// TIA Portal V20 export
FUNCTION "CallCycleTimerMapping" : Void   // FC32781, LAD
// stored: SetENOAutomatically false
   VAR CONSTANT
      TRUE : Bool := TRUE;
   END_VAR
BEGIN

REGION Network 1: cycleTimerDataSet[1]
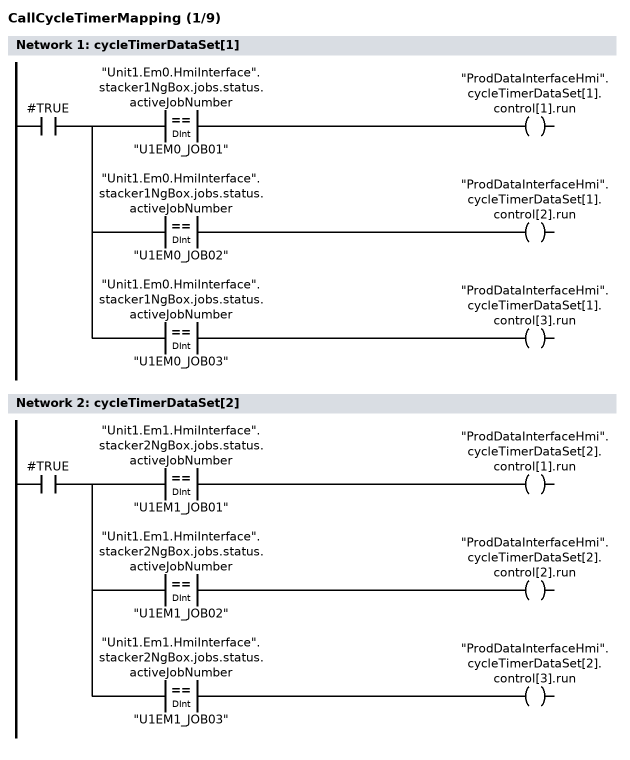
   RUNG wire#powerrail
      Contact( #TRUE )
      wire#w1
      { S7_Templates := "SrcType := DInt" } EQ_Contact(in1 := "Unit1.Em0.HmiInterface".stacker1NgBox.jobs.status.activeJobNumber, in2 := "U1EM0_JOB01")
      Coil( "ProdDataInterfaceHmi".cycleTimerDataSet[1].control[1].run )
   END_RUNG
   RUNG wire#w1
      { S7_Templates := "SrcType := DInt" } EQ_Contact(in1 := "Unit1.Em0.HmiInterface".stacker1NgBox.jobs.status.activeJobNumber, in2 := "U1EM0_JOB02")
      Coil( "ProdDataInterfaceHmi".cycleTimerDataSet[1].control[2].run )
   END_RUNG
   RUNG wire#w1
      { S7_Templates := "SrcType := DInt" } EQ_Contact(in1 := "Unit1.Em0.HmiInterface".stacker1NgBox.jobs.status.activeJobNumber, in2 := "U1EM0_JOB03")
      Coil( "ProdDataInterfaceHmi".cycleTimerDataSet[1].control[3].run )
   END_RUNG
   // the same network as SCL:
   "ProdDataInterfaceHmi".cycleTimerDataSet[1].control[1].run := #TRUE AND ("Unit1.Em0.HmiInterface".stacker1NgBox.jobs.status.activeJobNumber = "U1EM0_JOB01");
   "ProdDataInterfaceHmi".cycleTimerDataSet[1].control[2].run := #TRUE AND ("Unit1.Em0.HmiInterface".stacker1NgBox.jobs.status.activeJobNumber = "U1EM0_JOB02");
   "ProdDataInterfaceHmi".cycleTimerDataSet[1].control[3].run := #TRUE AND ("Unit1.Em0.HmiInterface".stacker1NgBox.jobs.status.activeJobNumber = "U1EM0_JOB03");
END_REGION

REGION Network 2: cycleTimerDataSet[2]
   RUNG wire#powerrail
      Contact( #TRUE )
      wire#w1
      { S7_Templates := "SrcType := DInt" } EQ_Contact(in1 := "Unit1.Em1.HmiInterface".stacker2NgBox.jobs.status.activeJobNumber, in2 := "U1EM1_JOB01")
      Coil( "ProdDataInterfaceHmi".cycleTimerDataSet[2].control[1].run )
   END_RUNG
   RUNG wire#w1
      { S7_Templates := "SrcType := DInt" } EQ_Contact(in1 := "Unit1.Em1.HmiInterface".stacker2NgBox.jobs.status.activeJobNumber, in2 := "U1EM1_JOB02")
      Coil( "ProdDataInterfaceHmi".cycleTimerDataSet[2].control[2].run )
   END_RUNG
   RUNG wire#w1
      { S7_Templates := "SrcType := DInt" } EQ_Contact(in1 := "Unit1.Em1.HmiInterface".stacker2NgBox.jobs.status.activeJobNumber, in2 := "U1EM1_JOB03")
      Coil( "ProdDataInterfaceHmi".cycleTimerDataSet[2].control[3].run )
   END_RUNG
   // the same network as SCL:
   "ProdDataInterfaceHmi".cycleTimerDataSet[2].control[1].run := #TRUE AND ("Unit1.Em1.HmiInterface".stacker2NgBox.jobs.status.activeJobNumber = "U1EM1_JOB01");
   "ProdDataInterfaceHmi".cycleTimerDataSet[2].control[2].run := #TRUE AND ("Unit1.Em1.HmiInterface".stacker2NgBox.jobs.status.activeJobNumber = "U1EM1_JOB02");
   "ProdDataInterfaceHmi".cycleTimerDataSet[2].control[3].run := #TRUE AND ("Unit1.Em1.HmiInterface".stacker2NgBox.jobs.status.activeJobNumber = "U1EM1_JOB03");
END_REGION

REGION Network 3: cycleTimerDataSet[3]
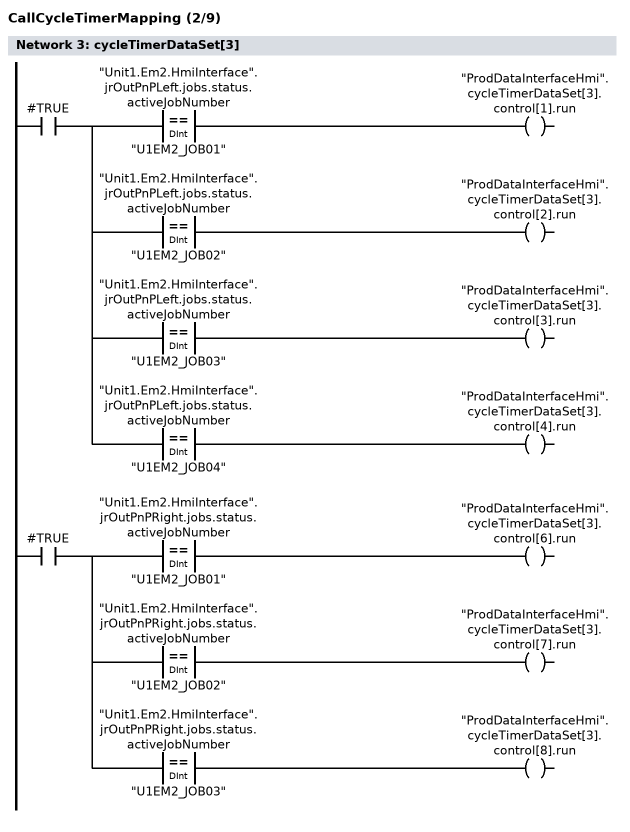
   RUNG wire#powerrail
      Contact( #TRUE )
      wire#w1
      { S7_Templates := "SrcType := DInt" } EQ_Contact(in1 := "Unit1.Em2.HmiInterface".jrOutPnPLeft.jobs.status.activeJobNumber, in2 := "U1EM2_JOB01")
      Coil( "ProdDataInterfaceHmi".cycleTimerDataSet[3].control[1].run )
   END_RUNG
   RUNG wire#w1
      { S7_Templates := "SrcType := DInt" } EQ_Contact(in1 := "Unit1.Em2.HmiInterface".jrOutPnPLeft.jobs.status.activeJobNumber, in2 := "U1EM2_JOB02")
      Coil( "ProdDataInterfaceHmi".cycleTimerDataSet[3].control[2].run )
   END_RUNG
   RUNG wire#w1
      { S7_Templates := "SrcType := DInt" } EQ_Contact(in1 := "Unit1.Em2.HmiInterface".jrOutPnPLeft.jobs.status.activeJobNumber, in2 := "U1EM2_JOB03")
      Coil( "ProdDataInterfaceHmi".cycleTimerDataSet[3].control[3].run )
   END_RUNG
   RUNG wire#w1
      { S7_Templates := "SrcType := DInt" } EQ_Contact(in1 := "Unit1.Em2.HmiInterface".jrOutPnPLeft.jobs.status.activeJobNumber, in2 := "U1EM2_JOB04")
      Coil( "ProdDataInterfaceHmi".cycleTimerDataSet[3].control[4].run )
   END_RUNG
   RUNG wire#powerrail
      Contact( #TRUE )
      wire#w2
      { S7_Templates := "SrcType := DInt" } EQ_Contact(in1 := "Unit1.Em2.HmiInterface".jrOutPnPRight.jobs.status.activeJobNumber, in2 := "U1EM2_JOB01")
      Coil( "ProdDataInterfaceHmi".cycleTimerDataSet[3].control[6].run )
   END_RUNG
   RUNG wire#w2
      { S7_Templates := "SrcType := DInt" } EQ_Contact(in1 := "Unit1.Em2.HmiInterface".jrOutPnPRight.jobs.status.activeJobNumber, in2 := "U1EM2_JOB02")
      Coil( "ProdDataInterfaceHmi".cycleTimerDataSet[3].control[7].run )
   END_RUNG
   RUNG wire#w2
      { S7_Templates := "SrcType := DInt" } EQ_Contact(in1 := "Unit1.Em2.HmiInterface".jrOutPnPRight.jobs.status.activeJobNumber, in2 := "U1EM2_JOB03")
      Coil( "ProdDataInterfaceHmi".cycleTimerDataSet[3].control[8].run )
   END_RUNG
   // the same network as SCL:
   "ProdDataInterfaceHmi".cycleTimerDataSet[3].control[1].run := #TRUE AND ("Unit1.Em2.HmiInterface".jrOutPnPLeft.jobs.status.activeJobNumber = "U1EM2_JOB01");
   "ProdDataInterfaceHmi".cycleTimerDataSet[3].control[2].run := #TRUE AND ("Unit1.Em2.HmiInterface".jrOutPnPLeft.jobs.status.activeJobNumber = "U1EM2_JOB02");
   "ProdDataInterfaceHmi".cycleTimerDataSet[3].control[3].run := #TRUE AND ("Unit1.Em2.HmiInterface".jrOutPnPLeft.jobs.status.activeJobNumber = "U1EM2_JOB03");
   "ProdDataInterfaceHmi".cycleTimerDataSet[3].control[4].run := #TRUE AND ("Unit1.Em2.HmiInterface".jrOutPnPLeft.jobs.status.activeJobNumber = "U1EM2_JOB04");
   "ProdDataInterfaceHmi".cycleTimerDataSet[3].control[6].run := #TRUE AND ("Unit1.Em2.HmiInterface".jrOutPnPRight.jobs.status.activeJobNumber = "U1EM2_JOB01");
   "ProdDataInterfaceHmi".cycleTimerDataSet[3].control[7].run := #TRUE AND ("Unit1.Em2.HmiInterface".jrOutPnPRight.jobs.status.activeJobNumber = "U1EM2_JOB02");
   "ProdDataInterfaceHmi".cycleTimerDataSet[3].control[8].run := #TRUE AND ("Unit1.Em2.HmiInterface".jrOutPnPRight.jobs.status.activeJobNumber = "U1EM2_JOB03");
END_REGION

REGION Network 4: cycleTimerDataSet[4]
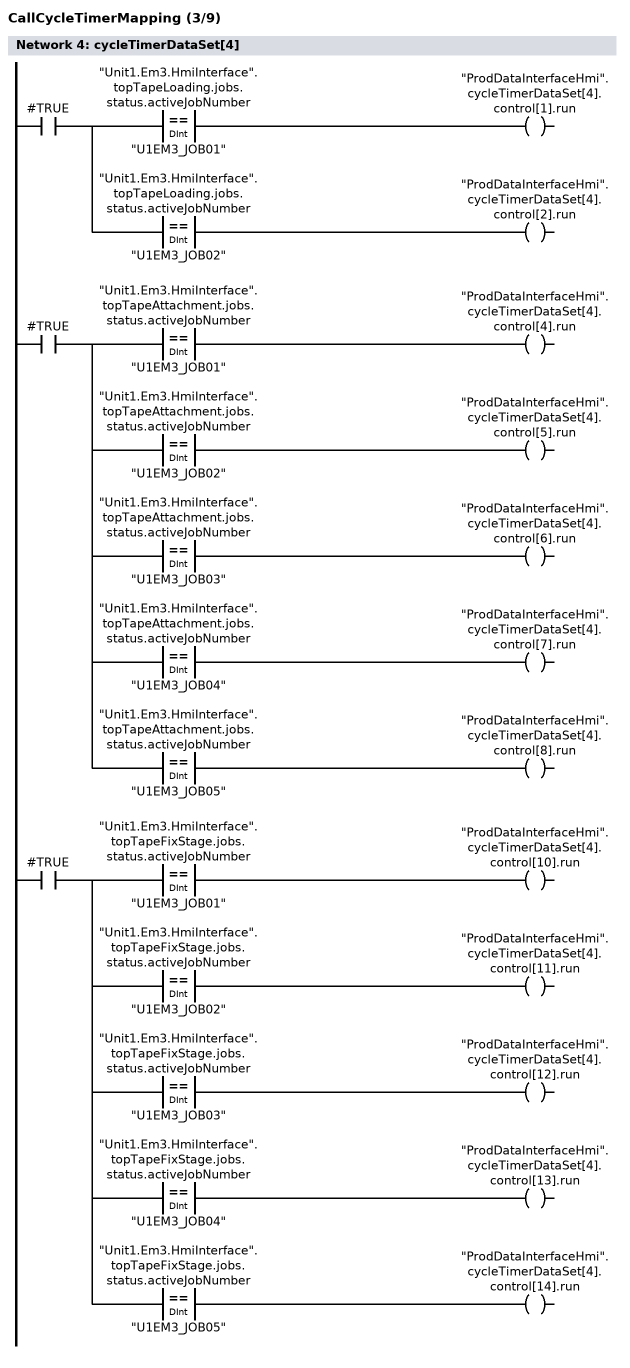
   RUNG wire#powerrail
      Contact( #TRUE )
      wire#w1
      { S7_Templates := "SrcType := DInt" } EQ_Contact(in1 := "Unit1.Em3.HmiInterface".topTapeLoading.jobs.status.activeJobNumber, in2 := "U1EM3_JOB01")
      Coil( "ProdDataInterfaceHmi".cycleTimerDataSet[4].control[1].run )
   END_RUNG
   RUNG wire#w1
      { S7_Templates := "SrcType := DInt" } EQ_Contact(in1 := "Unit1.Em3.HmiInterface".topTapeLoading.jobs.status.activeJobNumber, in2 := "U1EM3_JOB02")
      Coil( "ProdDataInterfaceHmi".cycleTimerDataSet[4].control[2].run )
   END_RUNG
   RUNG wire#powerrail
      Contact( #TRUE )
      wire#w2
      { S7_Templates := "SrcType := DInt" } EQ_Contact(in1 := "Unit1.Em3.HmiInterface".topTapeAttachment.jobs.status.activeJobNumber, in2 := "U1EM3_JOB01")
      Coil( "ProdDataInterfaceHmi".cycleTimerDataSet[4].control[4].run )
   END_RUNG
   RUNG wire#w2
      { S7_Templates := "SrcType := DInt" } EQ_Contact(in1 := "Unit1.Em3.HmiInterface".topTapeAttachment.jobs.status.activeJobNumber, in2 := "U1EM3_JOB02")
      Coil( "ProdDataInterfaceHmi".cycleTimerDataSet[4].control[5].run )
   END_RUNG
   RUNG wire#w2
      { S7_Templates := "SrcType := DInt" } EQ_Contact(in1 := "Unit1.Em3.HmiInterface".topTapeAttachment.jobs.status.activeJobNumber, in2 := "U1EM3_JOB03")
      Coil( "ProdDataInterfaceHmi".cycleTimerDataSet[4].control[6].run )
   END_RUNG
   RUNG wire#w2
      { S7_Templates := "SrcType := DInt" } EQ_Contact(in1 := "Unit1.Em3.HmiInterface".topTapeAttachment.jobs.status.activeJobNumber, in2 := "U1EM3_JOB04")
      Coil( "ProdDataInterfaceHmi".cycleTimerDataSet[4].control[7].run )
   END_RUNG
   RUNG wire#w2
      { S7_Templates := "SrcType := DInt" } EQ_Contact(in1 := "Unit1.Em3.HmiInterface".topTapeAttachment.jobs.status.activeJobNumber, in2 := "U1EM3_JOB05")
      Coil( "ProdDataInterfaceHmi".cycleTimerDataSet[4].control[8].run )
   END_RUNG
   RUNG wire#powerrail
      Contact( #TRUE )
      wire#w3
      { S7_Templates := "SrcType := DInt" } EQ_Contact(in1 := "Unit1.Em3.HmiInterface".topTapeFixStage.jobs.status.activeJobNumber, in2 := "U1EM3_JOB01")
      Coil( "ProdDataInterfaceHmi".cycleTimerDataSet[4].control[10].run )
   END_RUNG
   RUNG wire#w3
      { S7_Templates := "SrcType := DInt" } EQ_Contact(in1 := "Unit1.Em3.HmiInterface".topTapeFixStage.jobs.status.activeJobNumber, in2 := "U1EM3_JOB02")
      Coil( "ProdDataInterfaceHmi".cycleTimerDataSet[4].control[11].run )
   END_RUNG
   RUNG wire#w3
      { S7_Templates := "SrcType := DInt" } EQ_Contact(in1 := "Unit1.Em3.HmiInterface".topTapeFixStage.jobs.status.activeJobNumber, in2 := "U1EM3_JOB03")
      Coil( "ProdDataInterfaceHmi".cycleTimerDataSet[4].control[12].run )
   END_RUNG
   RUNG wire#w3
      { S7_Templates := "SrcType := DInt" } EQ_Contact(in1 := "Unit1.Em3.HmiInterface".topTapeFixStage.jobs.status.activeJobNumber, in2 := "U1EM3_JOB04")
      Coil( "ProdDataInterfaceHmi".cycleTimerDataSet[4].control[13].run )
   END_RUNG
   RUNG wire#w3
      { S7_Templates := "SrcType := DInt" } EQ_Contact(in1 := "Unit1.Em3.HmiInterface".topTapeFixStage.jobs.status.activeJobNumber, in2 := "U1EM3_JOB05")
      Coil( "ProdDataInterfaceHmi".cycleTimerDataSet[4].control[14].run )
   END_RUNG
   // the same network as SCL:
   "ProdDataInterfaceHmi".cycleTimerDataSet[4].control[1].run := #TRUE AND ("Unit1.Em3.HmiInterface".topTapeLoading.jobs.status.activeJobNumber = "U1EM3_JOB01");
   "ProdDataInterfaceHmi".cycleTimerDataSet[4].control[2].run := #TRUE AND ("Unit1.Em3.HmiInterface".topTapeLoading.jobs.status.activeJobNumber = "U1EM3_JOB02");
   "ProdDataInterfaceHmi".cycleTimerDataSet[4].control[4].run := #TRUE AND ("Unit1.Em3.HmiInterface".topTapeAttachment.jobs.status.activeJobNumber = "U1EM3_JOB01");
   "ProdDataInterfaceHmi".cycleTimerDataSet[4].control[5].run := #TRUE AND ("Unit1.Em3.HmiInterface".topTapeAttachment.jobs.status.activeJobNumber = "U1EM3_JOB02");
   "ProdDataInterfaceHmi".cycleTimerDataSet[4].control[6].run := #TRUE AND ("Unit1.Em3.HmiInterface".topTapeAttachment.jobs.status.activeJobNumber = "U1EM3_JOB03");
   "ProdDataInterfaceHmi".cycleTimerDataSet[4].control[7].run := #TRUE AND ("Unit1.Em3.HmiInterface".topTapeAttachment.jobs.status.activeJobNumber = "U1EM3_JOB04");
   "ProdDataInterfaceHmi".cycleTimerDataSet[4].control[8].run := #TRUE AND ("Unit1.Em3.HmiInterface".topTapeAttachment.jobs.status.activeJobNumber = "U1EM3_JOB05");
   "ProdDataInterfaceHmi".cycleTimerDataSet[4].control[10].run := #TRUE AND ("Unit1.Em3.HmiInterface".topTapeFixStage.jobs.status.activeJobNumber = "U1EM3_JOB01");
   "ProdDataInterfaceHmi".cycleTimerDataSet[4].control[11].run := #TRUE AND ("Unit1.Em3.HmiInterface".topTapeFixStage.jobs.status.activeJobNumber = "U1EM3_JOB02");
   "ProdDataInterfaceHmi".cycleTimerDataSet[4].control[12].run := #TRUE AND ("Unit1.Em3.HmiInterface".topTapeFixStage.jobs.status.activeJobNumber = "U1EM3_JOB03");
   "ProdDataInterfaceHmi".cycleTimerDataSet[4].control[13].run := #TRUE AND ("Unit1.Em3.HmiInterface".topTapeFixStage.jobs.status.activeJobNumber = "U1EM3_JOB04");
   "ProdDataInterfaceHmi".cycleTimerDataSet[4].control[14].run := #TRUE AND ("Unit1.Em3.HmiInterface".topTapeFixStage.jobs.status.activeJobNumber = "U1EM3_JOB05");
END_REGION

REGION Network 5: cycleTimerDataSet[5]
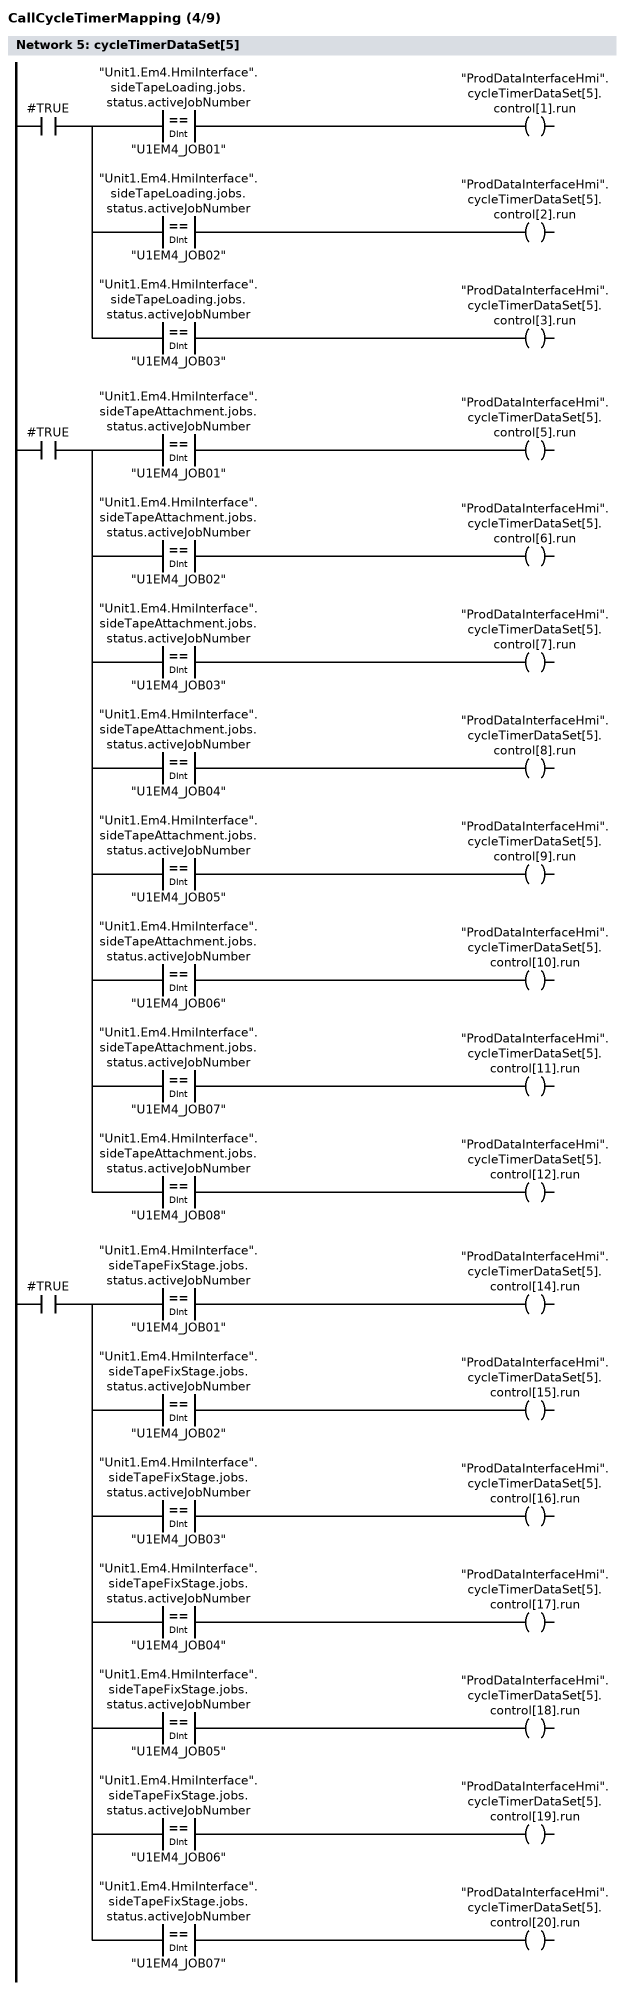
   RUNG wire#powerrail
      Contact( #TRUE )
      wire#w1
      { S7_Templates := "SrcType := DInt" } EQ_Contact(in1 := "Unit1.Em4.HmiInterface".sideTapeLoading.jobs.status.activeJobNumber, in2 := "U1EM4_JOB01")
      Coil( "ProdDataInterfaceHmi".cycleTimerDataSet[5].control[1].run )
   END_RUNG
   RUNG wire#w1
      { S7_Templates := "SrcType := DInt" } EQ_Contact(in1 := "Unit1.Em4.HmiInterface".sideTapeLoading.jobs.status.activeJobNumber, in2 := "U1EM4_JOB02")
      Coil( "ProdDataInterfaceHmi".cycleTimerDataSet[5].control[2].run )
   END_RUNG
   RUNG wire#w1
      { S7_Templates := "SrcType := DInt" } EQ_Contact(in1 := "Unit1.Em4.HmiInterface".sideTapeLoading.jobs.status.activeJobNumber, in2 := "U1EM4_JOB03")
      Coil( "ProdDataInterfaceHmi".cycleTimerDataSet[5].control[3].run )
   END_RUNG
   RUNG wire#powerrail
      Contact( #TRUE )
      wire#w2
      { S7_Templates := "SrcType := DInt" } EQ_Contact(in1 := "Unit1.Em4.HmiInterface".sideTapeAttachment.jobs.status.activeJobNumber, in2 := "U1EM4_JOB01")
      Coil( "ProdDataInterfaceHmi".cycleTimerDataSet[5].control[5].run )
   END_RUNG
   RUNG wire#w2
      { S7_Templates := "SrcType := DInt" } EQ_Contact(in1 := "Unit1.Em4.HmiInterface".sideTapeAttachment.jobs.status.activeJobNumber, in2 := "U1EM4_JOB02")
      Coil( "ProdDataInterfaceHmi".cycleTimerDataSet[5].control[6].run )
   END_RUNG
   RUNG wire#w2
      { S7_Templates := "SrcType := DInt" } EQ_Contact(in1 := "Unit1.Em4.HmiInterface".sideTapeAttachment.jobs.status.activeJobNumber, in2 := "U1EM4_JOB03")
      Coil( "ProdDataInterfaceHmi".cycleTimerDataSet[5].control[7].run )
   END_RUNG
   RUNG wire#w2
      { S7_Templates := "SrcType := DInt" } EQ_Contact(in1 := "Unit1.Em4.HmiInterface".sideTapeAttachment.jobs.status.activeJobNumber, in2 := "U1EM4_JOB04")
      Coil( "ProdDataInterfaceHmi".cycleTimerDataSet[5].control[8].run )
   END_RUNG
   RUNG wire#w2
      { S7_Templates := "SrcType := DInt" } EQ_Contact(in1 := "Unit1.Em4.HmiInterface".sideTapeAttachment.jobs.status.activeJobNumber, in2 := "U1EM4_JOB05")
      Coil( "ProdDataInterfaceHmi".cycleTimerDataSet[5].control[9].run )
   END_RUNG
   RUNG wire#w2
      { S7_Templates := "SrcType := DInt" } EQ_Contact(in1 := "Unit1.Em4.HmiInterface".sideTapeAttachment.jobs.status.activeJobNumber, in2 := "U1EM4_JOB06")
      Coil( "ProdDataInterfaceHmi".cycleTimerDataSet[5].control[10].run )
   END_RUNG
   RUNG wire#w2
      { S7_Templates := "SrcType := DInt" } EQ_Contact(in1 := "Unit1.Em4.HmiInterface".sideTapeAttachment.jobs.status.activeJobNumber, in2 := "U1EM4_JOB07")
      Coil( "ProdDataInterfaceHmi".cycleTimerDataSet[5].control[11].run )
   END_RUNG
   RUNG wire#w2
      { S7_Templates := "SrcType := DInt" } EQ_Contact(in1 := "Unit1.Em4.HmiInterface".sideTapeAttachment.jobs.status.activeJobNumber, in2 := "U1EM4_JOB08")
      Coil( "ProdDataInterfaceHmi".cycleTimerDataSet[5].control[12].run )
   END_RUNG
   RUNG wire#powerrail
      Contact( #TRUE )
      wire#w3
      { S7_Templates := "SrcType := DInt" } EQ_Contact(in1 := "Unit1.Em4.HmiInterface".sideTapeFixStage.jobs.status.activeJobNumber, in2 := "U1EM4_JOB01")
      Coil( "ProdDataInterfaceHmi".cycleTimerDataSet[5].control[14].run )
   END_RUNG
   RUNG wire#w3
      { S7_Templates := "SrcType := DInt" } EQ_Contact(in1 := "Unit1.Em4.HmiInterface".sideTapeFixStage.jobs.status.activeJobNumber, in2 := "U1EM4_JOB02")
      Coil( "ProdDataInterfaceHmi".cycleTimerDataSet[5].control[15].run )
   END_RUNG
   RUNG wire#w3
      { S7_Templates := "SrcType := DInt" } EQ_Contact(in1 := "Unit1.Em4.HmiInterface".sideTapeFixStage.jobs.status.activeJobNumber, in2 := "U1EM4_JOB03")
      Coil( "ProdDataInterfaceHmi".cycleTimerDataSet[5].control[16].run )
   END_RUNG
   RUNG wire#w3
      { S7_Templates := "SrcType := DInt" } EQ_Contact(in1 := "Unit1.Em4.HmiInterface".sideTapeFixStage.jobs.status.activeJobNumber, in2 := "U1EM4_JOB04")
      Coil( "ProdDataInterfaceHmi".cycleTimerDataSet[5].control[17].run )
   END_RUNG
   RUNG wire#w3
      { S7_Templates := "SrcType := DInt" } EQ_Contact(in1 := "Unit1.Em4.HmiInterface".sideTapeFixStage.jobs.status.activeJobNumber, in2 := "U1EM4_JOB05")
      Coil( "ProdDataInterfaceHmi".cycleTimerDataSet[5].control[18].run )
   END_RUNG
   RUNG wire#w3
      { S7_Templates := "SrcType := DInt" } EQ_Contact(in1 := "Unit1.Em4.HmiInterface".sideTapeFixStage.jobs.status.activeJobNumber, in2 := "U1EM4_JOB06")
      Coil( "ProdDataInterfaceHmi".cycleTimerDataSet[5].control[19].run )
   END_RUNG
   RUNG wire#w3
      { S7_Templates := "SrcType := DInt" } EQ_Contact(in1 := "Unit1.Em4.HmiInterface".sideTapeFixStage.jobs.status.activeJobNumber, in2 := "U1EM4_JOB07")
      Coil( "ProdDataInterfaceHmi".cycleTimerDataSet[5].control[20].run )
   END_RUNG
   // the same network as SCL:
   "ProdDataInterfaceHmi".cycleTimerDataSet[5].control[1].run := #TRUE AND ("Unit1.Em4.HmiInterface".sideTapeLoading.jobs.status.activeJobNumber = "U1EM4_JOB01");
   "ProdDataInterfaceHmi".cycleTimerDataSet[5].control[2].run := #TRUE AND ("Unit1.Em4.HmiInterface".sideTapeLoading.jobs.status.activeJobNumber = "U1EM4_JOB02");
   "ProdDataInterfaceHmi".cycleTimerDataSet[5].control[3].run := #TRUE AND ("Unit1.Em4.HmiInterface".sideTapeLoading.jobs.status.activeJobNumber = "U1EM4_JOB03");
   "ProdDataInterfaceHmi".cycleTimerDataSet[5].control[5].run := #TRUE AND ("Unit1.Em4.HmiInterface".sideTapeAttachment.jobs.status.activeJobNumber = "U1EM4_JOB01");
   "ProdDataInterfaceHmi".cycleTimerDataSet[5].control[6].run := #TRUE AND ("Unit1.Em4.HmiInterface".sideTapeAttachment.jobs.status.activeJobNumber = "U1EM4_JOB02");
   "ProdDataInterfaceHmi".cycleTimerDataSet[5].control[7].run := #TRUE AND ("Unit1.Em4.HmiInterface".sideTapeAttachment.jobs.status.activeJobNumber = "U1EM4_JOB03");
   "ProdDataInterfaceHmi".cycleTimerDataSet[5].control[8].run := #TRUE AND ("Unit1.Em4.HmiInterface".sideTapeAttachment.jobs.status.activeJobNumber = "U1EM4_JOB04");
   "ProdDataInterfaceHmi".cycleTimerDataSet[5].control[9].run := #TRUE AND ("Unit1.Em4.HmiInterface".sideTapeAttachment.jobs.status.activeJobNumber = "U1EM4_JOB05");
   "ProdDataInterfaceHmi".cycleTimerDataSet[5].control[10].run := #TRUE AND ("Unit1.Em4.HmiInterface".sideTapeAttachment.jobs.status.activeJobNumber = "U1EM4_JOB06");
   "ProdDataInterfaceHmi".cycleTimerDataSet[5].control[11].run := #TRUE AND ("Unit1.Em4.HmiInterface".sideTapeAttachment.jobs.status.activeJobNumber = "U1EM4_JOB07");
   "ProdDataInterfaceHmi".cycleTimerDataSet[5].control[12].run := #TRUE AND ("Unit1.Em4.HmiInterface".sideTapeAttachment.jobs.status.activeJobNumber = "U1EM4_JOB08");
   "ProdDataInterfaceHmi".cycleTimerDataSet[5].control[14].run := #TRUE AND ("Unit1.Em4.HmiInterface".sideTapeFixStage.jobs.status.activeJobNumber = "U1EM4_JOB01");
   "ProdDataInterfaceHmi".cycleTimerDataSet[5].control[15].run := #TRUE AND ("Unit1.Em4.HmiInterface".sideTapeFixStage.jobs.status.activeJobNumber = "U1EM4_JOB02");
   "ProdDataInterfaceHmi".cycleTimerDataSet[5].control[16].run := #TRUE AND ("Unit1.Em4.HmiInterface".sideTapeFixStage.jobs.status.activeJobNumber = "U1EM4_JOB03");
   "ProdDataInterfaceHmi".cycleTimerDataSet[5].control[17].run := #TRUE AND ("Unit1.Em4.HmiInterface".sideTapeFixStage.jobs.status.activeJobNumber = "U1EM4_JOB04");
   "ProdDataInterfaceHmi".cycleTimerDataSet[5].control[18].run := #TRUE AND ("Unit1.Em4.HmiInterface".sideTapeFixStage.jobs.status.activeJobNumber = "U1EM4_JOB05");
   "ProdDataInterfaceHmi".cycleTimerDataSet[5].control[19].run := #TRUE AND ("Unit1.Em4.HmiInterface".sideTapeFixStage.jobs.status.activeJobNumber = "U1EM4_JOB06");
   "ProdDataInterfaceHmi".cycleTimerDataSet[5].control[20].run := #TRUE AND ("Unit1.Em4.HmiInterface".sideTapeFixStage.jobs.status.activeJobNumber = "U1EM4_JOB07");
END_REGION

REGION Network 6: cycleTimerDataSet[6]
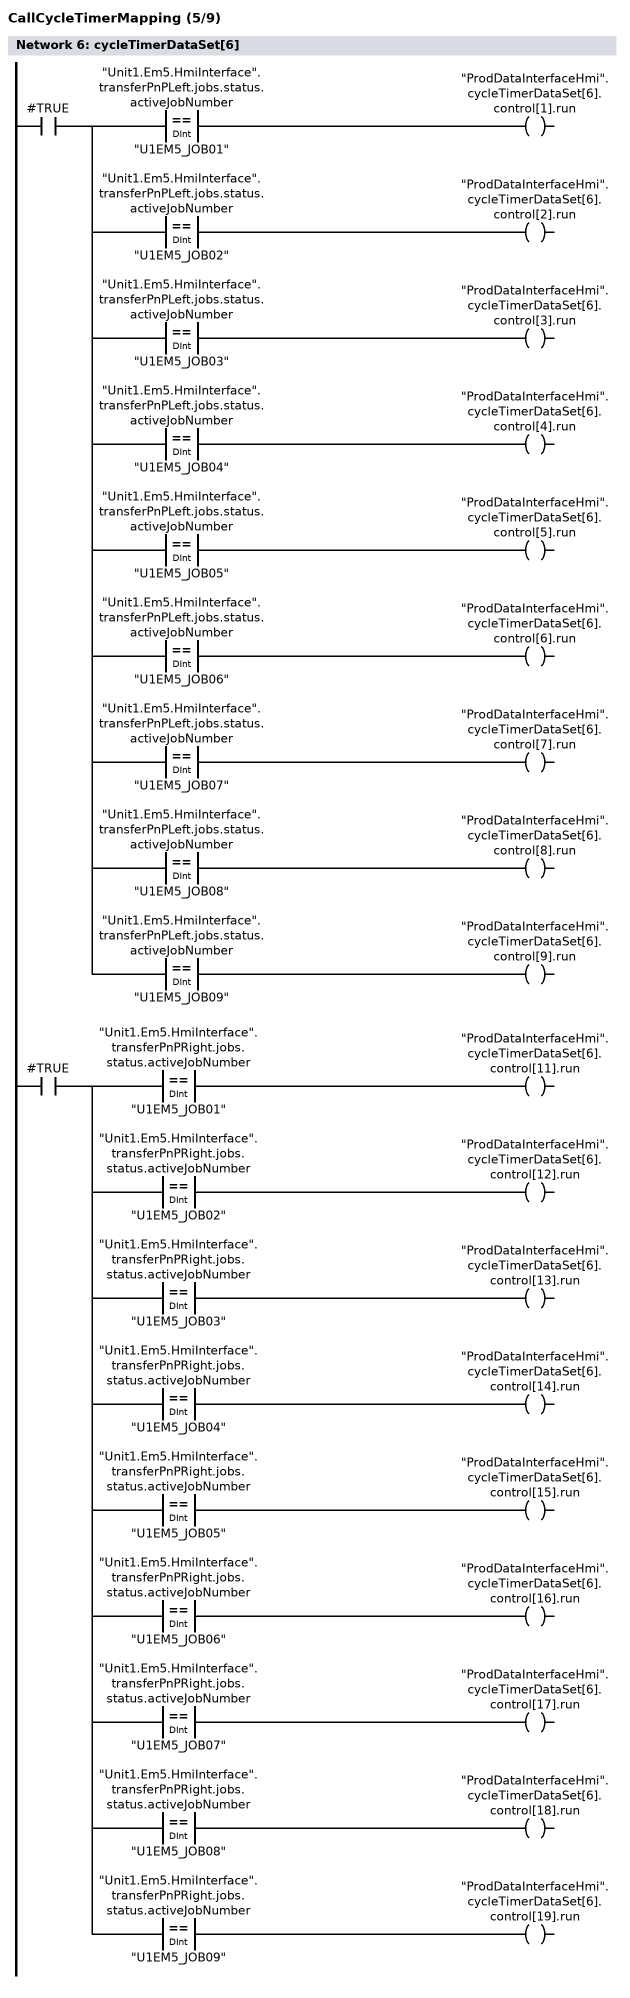
   RUNG wire#powerrail
      Contact( #TRUE )
      wire#w1
      { S7_Templates := "SrcType := DInt" } EQ_Contact(in1 := "Unit1.Em5.HmiInterface".transferPnPLeft.jobs.status.activeJobNumber, in2 := "U1EM5_JOB01")
      Coil( "ProdDataInterfaceHmi".cycleTimerDataSet[6].control[1].run )
   END_RUNG
   RUNG wire#w1
      { S7_Templates := "SrcType := DInt" } EQ_Contact(in1 := "Unit1.Em5.HmiInterface".transferPnPLeft.jobs.status.activeJobNumber, in2 := "U1EM5_JOB02")
      Coil( "ProdDataInterfaceHmi".cycleTimerDataSet[6].control[2].run )
   END_RUNG
   RUNG wire#w1
      { S7_Templates := "SrcType := DInt" } EQ_Contact(in1 := "Unit1.Em5.HmiInterface".transferPnPLeft.jobs.status.activeJobNumber, in2 := "U1EM5_JOB03")
      Coil( "ProdDataInterfaceHmi".cycleTimerDataSet[6].control[3].run )
   END_RUNG
   RUNG wire#w1
      { S7_Templates := "SrcType := DInt" } EQ_Contact(in1 := "Unit1.Em5.HmiInterface".transferPnPLeft.jobs.status.activeJobNumber, in2 := "U1EM5_JOB04")
      Coil( "ProdDataInterfaceHmi".cycleTimerDataSet[6].control[4].run )
   END_RUNG
   RUNG wire#w1
      { S7_Templates := "SrcType := DInt" } EQ_Contact(in1 := "Unit1.Em5.HmiInterface".transferPnPLeft.jobs.status.activeJobNumber, in2 := "U1EM5_JOB05")
      Coil( "ProdDataInterfaceHmi".cycleTimerDataSet[6].control[5].run )
   END_RUNG
   RUNG wire#w1
      { S7_Templates := "SrcType := DInt" } EQ_Contact(in1 := "Unit1.Em5.HmiInterface".transferPnPLeft.jobs.status.activeJobNumber, in2 := "U1EM5_JOB06")
      Coil( "ProdDataInterfaceHmi".cycleTimerDataSet[6].control[6].run )
   END_RUNG
   RUNG wire#w1
      { S7_Templates := "SrcType := DInt" } EQ_Contact(in1 := "Unit1.Em5.HmiInterface".transferPnPLeft.jobs.status.activeJobNumber, in2 := "U1EM5_JOB07")
      Coil( "ProdDataInterfaceHmi".cycleTimerDataSet[6].control[7].run )
   END_RUNG
   RUNG wire#w1
      { S7_Templates := "SrcType := DInt" } EQ_Contact(in1 := "Unit1.Em5.HmiInterface".transferPnPLeft.jobs.status.activeJobNumber, in2 := "U1EM5_JOB08")
      Coil( "ProdDataInterfaceHmi".cycleTimerDataSet[6].control[8].run )
   END_RUNG
   RUNG wire#w1
      { S7_Templates := "SrcType := DInt" } EQ_Contact(in1 := "Unit1.Em5.HmiInterface".transferPnPLeft.jobs.status.activeJobNumber, in2 := "U1EM5_JOB09")
      Coil( "ProdDataInterfaceHmi".cycleTimerDataSet[6].control[9].run )
   END_RUNG
   RUNG wire#powerrail
      Contact( #TRUE )
      wire#w2
      { S7_Templates := "SrcType := DInt" } EQ_Contact(in1 := "Unit1.Em5.HmiInterface".transferPnPRight.jobs.status.activeJobNumber, in2 := "U1EM5_JOB01")
      Coil( "ProdDataInterfaceHmi".cycleTimerDataSet[6].control[11].run )
   END_RUNG
   RUNG wire#w2
      { S7_Templates := "SrcType := DInt" } EQ_Contact(in1 := "Unit1.Em5.HmiInterface".transferPnPRight.jobs.status.activeJobNumber, in2 := "U1EM5_JOB02")
      Coil( "ProdDataInterfaceHmi".cycleTimerDataSet[6].control[12].run )
   END_RUNG
   RUNG wire#w2
      { S7_Templates := "SrcType := DInt" } EQ_Contact(in1 := "Unit1.Em5.HmiInterface".transferPnPRight.jobs.status.activeJobNumber, in2 := "U1EM5_JOB03")
      Coil( "ProdDataInterfaceHmi".cycleTimerDataSet[6].control[13].run )
   END_RUNG
   RUNG wire#w2
      { S7_Templates := "SrcType := DInt" } EQ_Contact(in1 := "Unit1.Em5.HmiInterface".transferPnPRight.jobs.status.activeJobNumber, in2 := "U1EM5_JOB04")
      Coil( "ProdDataInterfaceHmi".cycleTimerDataSet[6].control[14].run )
   END_RUNG
   RUNG wire#w2
      { S7_Templates := "SrcType := DInt" } EQ_Contact(in1 := "Unit1.Em5.HmiInterface".transferPnPRight.jobs.status.activeJobNumber, in2 := "U1EM5_JOB05")
      Coil( "ProdDataInterfaceHmi".cycleTimerDataSet[6].control[15].run )
   END_RUNG
   RUNG wire#w2
      { S7_Templates := "SrcType := DInt" } EQ_Contact(in1 := "Unit1.Em5.HmiInterface".transferPnPRight.jobs.status.activeJobNumber, in2 := "U1EM5_JOB06")
      Coil( "ProdDataInterfaceHmi".cycleTimerDataSet[6].control[16].run )
   END_RUNG
   RUNG wire#w2
      { S7_Templates := "SrcType := DInt" } EQ_Contact(in1 := "Unit1.Em5.HmiInterface".transferPnPRight.jobs.status.activeJobNumber, in2 := "U1EM5_JOB07")
      Coil( "ProdDataInterfaceHmi".cycleTimerDataSet[6].control[17].run )
   END_RUNG
   RUNG wire#w2
      { S7_Templates := "SrcType := DInt" } EQ_Contact(in1 := "Unit1.Em5.HmiInterface".transferPnPRight.jobs.status.activeJobNumber, in2 := "U1EM5_JOB08")
      Coil( "ProdDataInterfaceHmi".cycleTimerDataSet[6].control[18].run )
   END_RUNG
   RUNG wire#w2
      { S7_Templates := "SrcType := DInt" } EQ_Contact(in1 := "Unit1.Em5.HmiInterface".transferPnPRight.jobs.status.activeJobNumber, in2 := "U1EM5_JOB09")
      Coil( "ProdDataInterfaceHmi".cycleTimerDataSet[6].control[19].run )
   END_RUNG
   // the same network as SCL:
   "ProdDataInterfaceHmi".cycleTimerDataSet[6].control[1].run := #TRUE AND ("Unit1.Em5.HmiInterface".transferPnPLeft.jobs.status.activeJobNumber = "U1EM5_JOB01");
   "ProdDataInterfaceHmi".cycleTimerDataSet[6].control[2].run := #TRUE AND ("Unit1.Em5.HmiInterface".transferPnPLeft.jobs.status.activeJobNumber = "U1EM5_JOB02");
   "ProdDataInterfaceHmi".cycleTimerDataSet[6].control[3].run := #TRUE AND ("Unit1.Em5.HmiInterface".transferPnPLeft.jobs.status.activeJobNumber = "U1EM5_JOB03");
   "ProdDataInterfaceHmi".cycleTimerDataSet[6].control[4].run := #TRUE AND ("Unit1.Em5.HmiInterface".transferPnPLeft.jobs.status.activeJobNumber = "U1EM5_JOB04");
   "ProdDataInterfaceHmi".cycleTimerDataSet[6].control[5].run := #TRUE AND ("Unit1.Em5.HmiInterface".transferPnPLeft.jobs.status.activeJobNumber = "U1EM5_JOB05");
   "ProdDataInterfaceHmi".cycleTimerDataSet[6].control[6].run := #TRUE AND ("Unit1.Em5.HmiInterface".transferPnPLeft.jobs.status.activeJobNumber = "U1EM5_JOB06");
   "ProdDataInterfaceHmi".cycleTimerDataSet[6].control[7].run := #TRUE AND ("Unit1.Em5.HmiInterface".transferPnPLeft.jobs.status.activeJobNumber = "U1EM5_JOB07");
   "ProdDataInterfaceHmi".cycleTimerDataSet[6].control[8].run := #TRUE AND ("Unit1.Em5.HmiInterface".transferPnPLeft.jobs.status.activeJobNumber = "U1EM5_JOB08");
   "ProdDataInterfaceHmi".cycleTimerDataSet[6].control[9].run := #TRUE AND ("Unit1.Em5.HmiInterface".transferPnPLeft.jobs.status.activeJobNumber = "U1EM5_JOB09");
   "ProdDataInterfaceHmi".cycleTimerDataSet[6].control[11].run := #TRUE AND ("Unit1.Em5.HmiInterface".transferPnPRight.jobs.status.activeJobNumber = "U1EM5_JOB01");
   "ProdDataInterfaceHmi".cycleTimerDataSet[6].control[12].run := #TRUE AND ("Unit1.Em5.HmiInterface".transferPnPRight.jobs.status.activeJobNumber = "U1EM5_JOB02");
   "ProdDataInterfaceHmi".cycleTimerDataSet[6].control[13].run := #TRUE AND ("Unit1.Em5.HmiInterface".transferPnPRight.jobs.status.activeJobNumber = "U1EM5_JOB03");
   "ProdDataInterfaceHmi".cycleTimerDataSet[6].control[14].run := #TRUE AND ("Unit1.Em5.HmiInterface".transferPnPRight.jobs.status.activeJobNumber = "U1EM5_JOB04");
   "ProdDataInterfaceHmi".cycleTimerDataSet[6].control[15].run := #TRUE AND ("Unit1.Em5.HmiInterface".transferPnPRight.jobs.status.activeJobNumber = "U1EM5_JOB05");
   "ProdDataInterfaceHmi".cycleTimerDataSet[6].control[16].run := #TRUE AND ("Unit1.Em5.HmiInterface".transferPnPRight.jobs.status.activeJobNumber = "U1EM5_JOB06");
   "ProdDataInterfaceHmi".cycleTimerDataSet[6].control[17].run := #TRUE AND ("Unit1.Em5.HmiInterface".transferPnPRight.jobs.status.activeJobNumber = "U1EM5_JOB07");
   "ProdDataInterfaceHmi".cycleTimerDataSet[6].control[18].run := #TRUE AND ("Unit1.Em5.HmiInterface".transferPnPRight.jobs.status.activeJobNumber = "U1EM5_JOB08");
   "ProdDataInterfaceHmi".cycleTimerDataSet[6].control[19].run := #TRUE AND ("Unit1.Em5.HmiInterface".transferPnPRight.jobs.status.activeJobNumber = "U1EM5_JOB09");
END_REGION

REGION Network 7: cycleTimerDataSet[7]
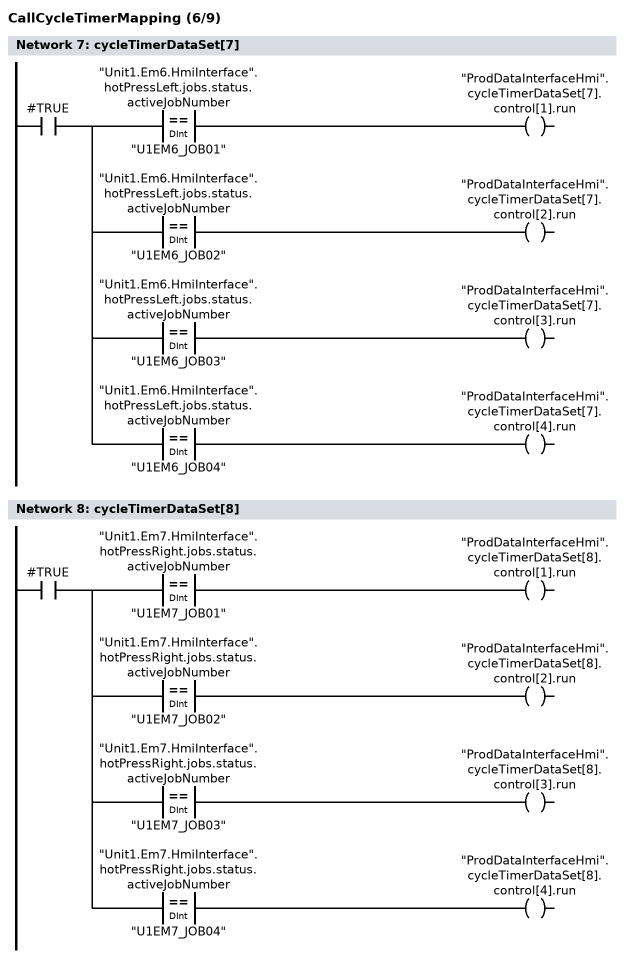
   RUNG wire#powerrail
      Contact( #TRUE )
      wire#w1
      { S7_Templates := "SrcType := DInt" } EQ_Contact(in1 := "Unit1.Em6.HmiInterface".hotPressLeft.jobs.status.activeJobNumber, in2 := "U1EM6_JOB01")
      Coil( "ProdDataInterfaceHmi".cycleTimerDataSet[7].control[1].run )
   END_RUNG
   RUNG wire#w1
      { S7_Templates := "SrcType := DInt" } EQ_Contact(in1 := "Unit1.Em6.HmiInterface".hotPressLeft.jobs.status.activeJobNumber, in2 := "U1EM6_JOB02")
      Coil( "ProdDataInterfaceHmi".cycleTimerDataSet[7].control[2].run )
   END_RUNG
   RUNG wire#w1
      { S7_Templates := "SrcType := DInt" } EQ_Contact(in1 := "Unit1.Em6.HmiInterface".hotPressLeft.jobs.status.activeJobNumber, in2 := "U1EM6_JOB03")
      Coil( "ProdDataInterfaceHmi".cycleTimerDataSet[7].control[3].run )
   END_RUNG
   RUNG wire#w1
      { S7_Templates := "SrcType := DInt" } EQ_Contact(in1 := "Unit1.Em6.HmiInterface".hotPressLeft.jobs.status.activeJobNumber, in2 := "U1EM6_JOB04")
      Coil( "ProdDataInterfaceHmi".cycleTimerDataSet[7].control[4].run )
   END_RUNG
   // the same network as SCL:
   "ProdDataInterfaceHmi".cycleTimerDataSet[7].control[1].run := #TRUE AND ("Unit1.Em6.HmiInterface".hotPressLeft.jobs.status.activeJobNumber = "U1EM6_JOB01");
   "ProdDataInterfaceHmi".cycleTimerDataSet[7].control[2].run := #TRUE AND ("Unit1.Em6.HmiInterface".hotPressLeft.jobs.status.activeJobNumber = "U1EM6_JOB02");
   "ProdDataInterfaceHmi".cycleTimerDataSet[7].control[3].run := #TRUE AND ("Unit1.Em6.HmiInterface".hotPressLeft.jobs.status.activeJobNumber = "U1EM6_JOB03");
   "ProdDataInterfaceHmi".cycleTimerDataSet[7].control[4].run := #TRUE AND ("Unit1.Em6.HmiInterface".hotPressLeft.jobs.status.activeJobNumber = "U1EM6_JOB04");
END_REGION

REGION Network 8: cycleTimerDataSet[8]
   RUNG wire#powerrail
      Contact( #TRUE )
      wire#w1
      { S7_Templates := "SrcType := DInt" } EQ_Contact(in1 := "Unit1.Em7.HmiInterface".hotPressRight.jobs.status.activeJobNumber, in2 := "U1EM7_JOB01")
      Coil( "ProdDataInterfaceHmi".cycleTimerDataSet[8].control[1].run )
   END_RUNG
   RUNG wire#w1
      { S7_Templates := "SrcType := DInt" } EQ_Contact(in1 := "Unit1.Em7.HmiInterface".hotPressRight.jobs.status.activeJobNumber, in2 := "U1EM7_JOB02")
      Coil( "ProdDataInterfaceHmi".cycleTimerDataSet[8].control[2].run )
   END_RUNG
   RUNG wire#w1
      { S7_Templates := "SrcType := DInt" } EQ_Contact(in1 := "Unit1.Em7.HmiInterface".hotPressRight.jobs.status.activeJobNumber, in2 := "U1EM7_JOB03")
      Coil( "ProdDataInterfaceHmi".cycleTimerDataSet[8].control[3].run )
   END_RUNG
   RUNG wire#w1
      { S7_Templates := "SrcType := DInt" } EQ_Contact(in1 := "Unit1.Em7.HmiInterface".hotPressRight.jobs.status.activeJobNumber, in2 := "U1EM7_JOB04")
      Coil( "ProdDataInterfaceHmi".cycleTimerDataSet[8].control[4].run )
   END_RUNG
   // the same network as SCL:
   "ProdDataInterfaceHmi".cycleTimerDataSet[8].control[1].run := #TRUE AND ("Unit1.Em7.HmiInterface".hotPressRight.jobs.status.activeJobNumber = "U1EM7_JOB01");
   "ProdDataInterfaceHmi".cycleTimerDataSet[8].control[2].run := #TRUE AND ("Unit1.Em7.HmiInterface".hotPressRight.jobs.status.activeJobNumber = "U1EM7_JOB02");
   "ProdDataInterfaceHmi".cycleTimerDataSet[8].control[3].run := #TRUE AND ("Unit1.Em7.HmiInterface".hotPressRight.jobs.status.activeJobNumber = "U1EM7_JOB03");
   "ProdDataInterfaceHmi".cycleTimerDataSet[8].control[4].run := #TRUE AND ("Unit1.Em7.HmiInterface".hotPressRight.jobs.status.activeJobNumber = "U1EM7_JOB04");
END_REGION

REGION Network 9: cycleTimerDataSet[9]
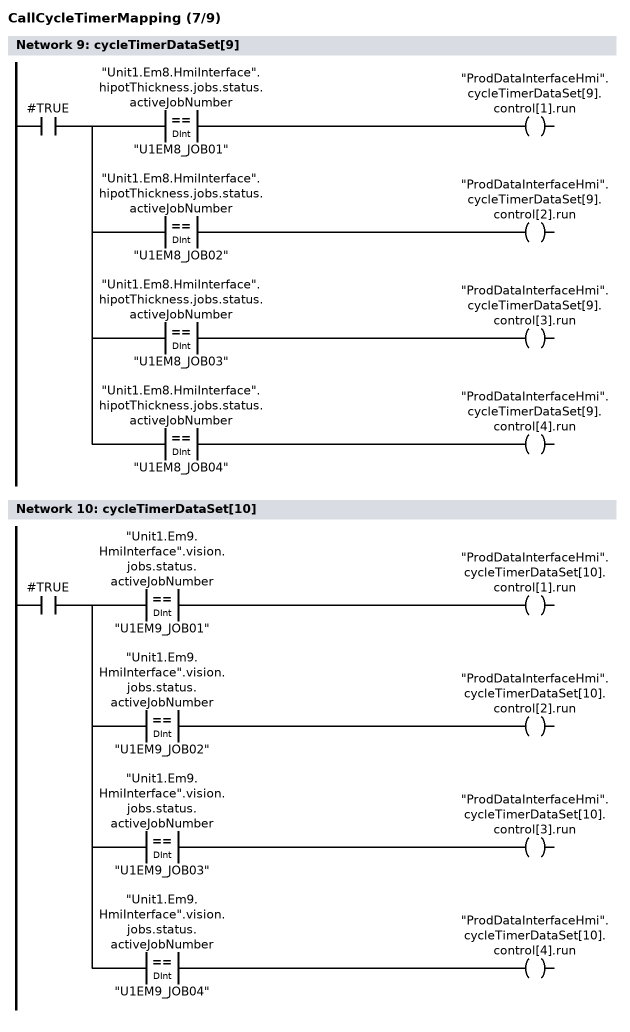
   RUNG wire#powerrail
      Contact( #TRUE )
      wire#w1
      { S7_Templates := "SrcType := DInt" } EQ_Contact(in1 := "Unit1.Em8.HmiInterface".hipotThickness.jobs.status.activeJobNumber, in2 := "U1EM8_JOB01")
      Coil( "ProdDataInterfaceHmi".cycleTimerDataSet[9].control[1].run )
   END_RUNG
   RUNG wire#w1
      { S7_Templates := "SrcType := DInt" } EQ_Contact(in1 := "Unit1.Em8.HmiInterface".hipotThickness.jobs.status.activeJobNumber, in2 := "U1EM8_JOB02")
      Coil( "ProdDataInterfaceHmi".cycleTimerDataSet[9].control[2].run )
   END_RUNG
   RUNG wire#w1
      { S7_Templates := "SrcType := DInt" } EQ_Contact(in1 := "Unit1.Em8.HmiInterface".hipotThickness.jobs.status.activeJobNumber, in2 := "U1EM8_JOB03")
      Coil( "ProdDataInterfaceHmi".cycleTimerDataSet[9].control[3].run )
   END_RUNG
   RUNG wire#w1
      { S7_Templates := "SrcType := DInt" } EQ_Contact(in1 := "Unit1.Em8.HmiInterface".hipotThickness.jobs.status.activeJobNumber, in2 := "U1EM8_JOB04")
      Coil( "ProdDataInterfaceHmi".cycleTimerDataSet[9].control[4].run )
   END_RUNG
   // the same network as SCL:
   "ProdDataInterfaceHmi".cycleTimerDataSet[9].control[1].run := #TRUE AND ("Unit1.Em8.HmiInterface".hipotThickness.jobs.status.activeJobNumber = "U1EM8_JOB01");
   "ProdDataInterfaceHmi".cycleTimerDataSet[9].control[2].run := #TRUE AND ("Unit1.Em8.HmiInterface".hipotThickness.jobs.status.activeJobNumber = "U1EM8_JOB02");
   "ProdDataInterfaceHmi".cycleTimerDataSet[9].control[3].run := #TRUE AND ("Unit1.Em8.HmiInterface".hipotThickness.jobs.status.activeJobNumber = "U1EM8_JOB03");
   "ProdDataInterfaceHmi".cycleTimerDataSet[9].control[4].run := #TRUE AND ("Unit1.Em8.HmiInterface".hipotThickness.jobs.status.activeJobNumber = "U1EM8_JOB04");
END_REGION

REGION Network 10: cycleTimerDataSet[10]
   RUNG wire#powerrail
      Contact( #TRUE )
      wire#w1
      { S7_Templates := "SrcType := DInt" } EQ_Contact(in1 := "Unit1.Em9.HmiInterface".vision.jobs.status.activeJobNumber, in2 := "U1EM9_JOB01")
      Coil( "ProdDataInterfaceHmi".cycleTimerDataSet[10].control[1].run )
   END_RUNG
   RUNG wire#w1
      { S7_Templates := "SrcType := DInt" } EQ_Contact(in1 := "Unit1.Em9.HmiInterface".vision.jobs.status.activeJobNumber, in2 := "U1EM9_JOB02")
      Coil( "ProdDataInterfaceHmi".cycleTimerDataSet[10].control[2].run )
   END_RUNG
   RUNG wire#w1
      { S7_Templates := "SrcType := DInt" } EQ_Contact(in1 := "Unit1.Em9.HmiInterface".vision.jobs.status.activeJobNumber, in2 := "U1EM9_JOB03")
      Coil( "ProdDataInterfaceHmi".cycleTimerDataSet[10].control[3].run )
   END_RUNG
   RUNG wire#w1
      { S7_Templates := "SrcType := DInt" } EQ_Contact(in1 := "Unit1.Em9.HmiInterface".vision.jobs.status.activeJobNumber, in2 := "U1EM9_JOB04")
      Coil( "ProdDataInterfaceHmi".cycleTimerDataSet[10].control[4].run )
   END_RUNG
   // the same network as SCL:
   "ProdDataInterfaceHmi".cycleTimerDataSet[10].control[1].run := #TRUE AND ("Unit1.Em9.HmiInterface".vision.jobs.status.activeJobNumber = "U1EM9_JOB01");
   "ProdDataInterfaceHmi".cycleTimerDataSet[10].control[2].run := #TRUE AND ("Unit1.Em9.HmiInterface".vision.jobs.status.activeJobNumber = "U1EM9_JOB02");
   "ProdDataInterfaceHmi".cycleTimerDataSet[10].control[3].run := #TRUE AND ("Unit1.Em9.HmiInterface".vision.jobs.status.activeJobNumber = "U1EM9_JOB03");
   "ProdDataInterfaceHmi".cycleTimerDataSet[10].control[4].run := #TRUE AND ("Unit1.Em9.HmiInterface".vision.jobs.status.activeJobNumber = "U1EM9_JOB04");
END_REGION

REGION Network 11: cycleTimerDataSet[11]
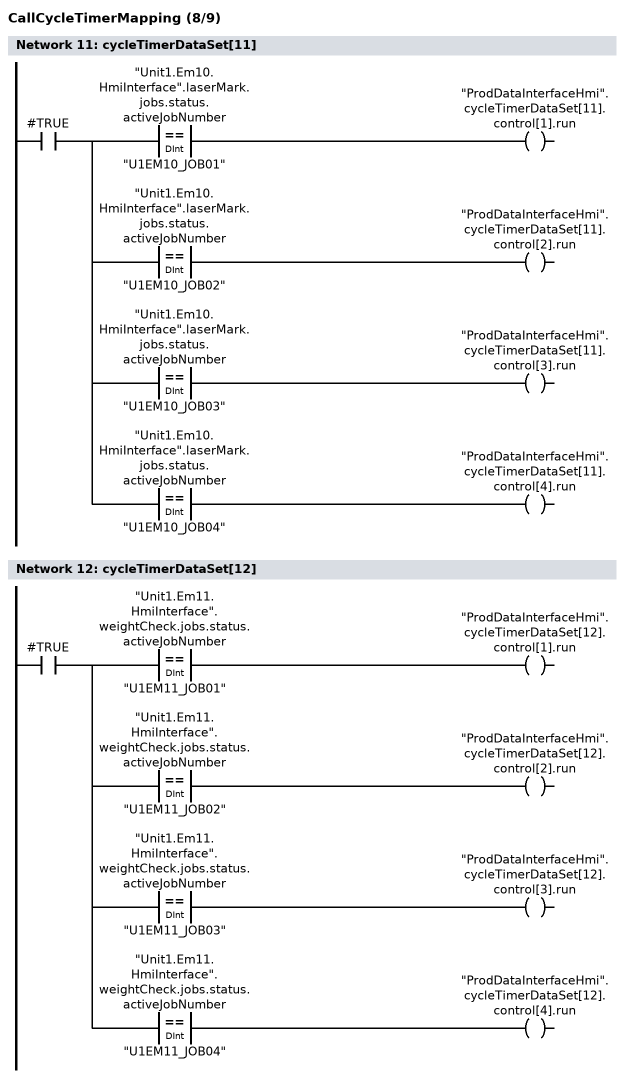
   RUNG wire#powerrail
      Contact( #TRUE )
      wire#w1
      { S7_Templates := "SrcType := DInt" } EQ_Contact(in1 := "Unit1.Em10.HmiInterface".laserMark.jobs.status.activeJobNumber, in2 := "U1EM10_JOB01")
      Coil( "ProdDataInterfaceHmi".cycleTimerDataSet[11].control[1].run )
   END_RUNG
   RUNG wire#w1
      { S7_Templates := "SrcType := DInt" } EQ_Contact(in1 := "Unit1.Em10.HmiInterface".laserMark.jobs.status.activeJobNumber, in2 := "U1EM10_JOB02")
      Coil( "ProdDataInterfaceHmi".cycleTimerDataSet[11].control[2].run )
   END_RUNG
   RUNG wire#w1
      { S7_Templates := "SrcType := DInt" } EQ_Contact(in1 := "Unit1.Em10.HmiInterface".laserMark.jobs.status.activeJobNumber, in2 := "U1EM10_JOB03")
      Coil( "ProdDataInterfaceHmi".cycleTimerDataSet[11].control[3].run )
   END_RUNG
   RUNG wire#w1
      { S7_Templates := "SrcType := DInt" } EQ_Contact(in1 := "Unit1.Em10.HmiInterface".laserMark.jobs.status.activeJobNumber, in2 := "U1EM10_JOB04")
      Coil( "ProdDataInterfaceHmi".cycleTimerDataSet[11].control[4].run )
   END_RUNG
   // the same network as SCL:
   "ProdDataInterfaceHmi".cycleTimerDataSet[11].control[1].run := #TRUE AND ("Unit1.Em10.HmiInterface".laserMark.jobs.status.activeJobNumber = "U1EM10_JOB01");
   "ProdDataInterfaceHmi".cycleTimerDataSet[11].control[2].run := #TRUE AND ("Unit1.Em10.HmiInterface".laserMark.jobs.status.activeJobNumber = "U1EM10_JOB02");
   "ProdDataInterfaceHmi".cycleTimerDataSet[11].control[3].run := #TRUE AND ("Unit1.Em10.HmiInterface".laserMark.jobs.status.activeJobNumber = "U1EM10_JOB03");
   "ProdDataInterfaceHmi".cycleTimerDataSet[11].control[4].run := #TRUE AND ("Unit1.Em10.HmiInterface".laserMark.jobs.status.activeJobNumber = "U1EM10_JOB04");
END_REGION

REGION Network 12: cycleTimerDataSet[12]
   RUNG wire#powerrail
      Contact( #TRUE )
      wire#w1
      { S7_Templates := "SrcType := DInt" } EQ_Contact(in1 := "Unit1.Em11.HmiInterface".weightCheck.jobs.status.activeJobNumber, in2 := "U1EM11_JOB01")
      Coil( "ProdDataInterfaceHmi".cycleTimerDataSet[12].control[1].run )
   END_RUNG
   RUNG wire#w1
      { S7_Templates := "SrcType := DInt" } EQ_Contact(in1 := "Unit1.Em11.HmiInterface".weightCheck.jobs.status.activeJobNumber, in2 := "U1EM11_JOB02")
      Coil( "ProdDataInterfaceHmi".cycleTimerDataSet[12].control[2].run )
   END_RUNG
   RUNG wire#w1
      { S7_Templates := "SrcType := DInt" } EQ_Contact(in1 := "Unit1.Em11.HmiInterface".weightCheck.jobs.status.activeJobNumber, in2 := "U1EM11_JOB03")
      Coil( "ProdDataInterfaceHmi".cycleTimerDataSet[12].control[3].run )
   END_RUNG
   RUNG wire#w1
      { S7_Templates := "SrcType := DInt" } EQ_Contact(in1 := "Unit1.Em11.HmiInterface".weightCheck.jobs.status.activeJobNumber, in2 := "U1EM11_JOB04")
      Coil( "ProdDataInterfaceHmi".cycleTimerDataSet[12].control[4].run )
   END_RUNG
   // the same network as SCL:
   "ProdDataInterfaceHmi".cycleTimerDataSet[12].control[1].run := #TRUE AND ("Unit1.Em11.HmiInterface".weightCheck.jobs.status.activeJobNumber = "U1EM11_JOB01");
   "ProdDataInterfaceHmi".cycleTimerDataSet[12].control[2].run := #TRUE AND ("Unit1.Em11.HmiInterface".weightCheck.jobs.status.activeJobNumber = "U1EM11_JOB02");
   "ProdDataInterfaceHmi".cycleTimerDataSet[12].control[3].run := #TRUE AND ("Unit1.Em11.HmiInterface".weightCheck.jobs.status.activeJobNumber = "U1EM11_JOB03");
   "ProdDataInterfaceHmi".cycleTimerDataSet[12].control[4].run := #TRUE AND ("Unit1.Em11.HmiInterface".weightCheck.jobs.status.activeJobNumber = "U1EM11_JOB04");
END_REGION

REGION Network 13: cycleTimerDataSet[13]
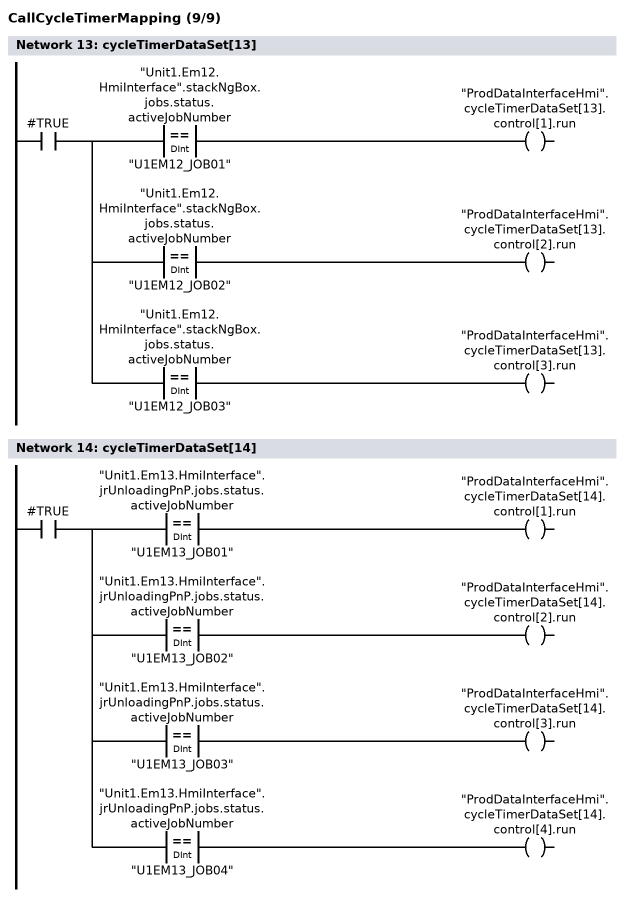
   RUNG wire#powerrail
      Contact( #TRUE )
      wire#w1
      { S7_Templates := "SrcType := DInt" } EQ_Contact(in1 := "Unit1.Em12.HmiInterface".stackNgBox.jobs.status.activeJobNumber, in2 := "U1EM12_JOB01")
      Coil( "ProdDataInterfaceHmi".cycleTimerDataSet[13].control[1].run )
   END_RUNG
   RUNG wire#w1
      { S7_Templates := "SrcType := DInt" } EQ_Contact(in1 := "Unit1.Em12.HmiInterface".stackNgBox.jobs.status.activeJobNumber, in2 := "U1EM12_JOB02")
      Coil( "ProdDataInterfaceHmi".cycleTimerDataSet[13].control[2].run )
   END_RUNG
   RUNG wire#w1
      { S7_Templates := "SrcType := DInt" } EQ_Contact(in1 := "Unit1.Em12.HmiInterface".stackNgBox.jobs.status.activeJobNumber, in2 := "U1EM12_JOB03")
      Coil( "ProdDataInterfaceHmi".cycleTimerDataSet[13].control[3].run )
   END_RUNG
   // the same network as SCL:
   "ProdDataInterfaceHmi".cycleTimerDataSet[13].control[1].run := #TRUE AND ("Unit1.Em12.HmiInterface".stackNgBox.jobs.status.activeJobNumber = "U1EM12_JOB01");
   "ProdDataInterfaceHmi".cycleTimerDataSet[13].control[2].run := #TRUE AND ("Unit1.Em12.HmiInterface".stackNgBox.jobs.status.activeJobNumber = "U1EM12_JOB02");
   "ProdDataInterfaceHmi".cycleTimerDataSet[13].control[3].run := #TRUE AND ("Unit1.Em12.HmiInterface".stackNgBox.jobs.status.activeJobNumber = "U1EM12_JOB03");
END_REGION

REGION Network 14: cycleTimerDataSet[14]
   RUNG wire#powerrail
      Contact( #TRUE )
      wire#w1
      { S7_Templates := "SrcType := DInt" } EQ_Contact(in1 := "Unit1.Em13.HmiInterface".jrUnloadingPnP.jobs.status.activeJobNumber, in2 := "U1EM13_JOB01")
      Coil( "ProdDataInterfaceHmi".cycleTimerDataSet[14].control[1].run )
   END_RUNG
   RUNG wire#w1
      { S7_Templates := "SrcType := DInt" } EQ_Contact(in1 := "Unit1.Em13.HmiInterface".jrUnloadingPnP.jobs.status.activeJobNumber, in2 := "U1EM13_JOB02")
      Coil( "ProdDataInterfaceHmi".cycleTimerDataSet[14].control[2].run )
   END_RUNG
   RUNG wire#w1
      { S7_Templates := "SrcType := DInt" } EQ_Contact(in1 := "Unit1.Em13.HmiInterface".jrUnloadingPnP.jobs.status.activeJobNumber, in2 := "U1EM13_JOB03")
      Coil( "ProdDataInterfaceHmi".cycleTimerDataSet[14].control[3].run )
   END_RUNG
   RUNG wire#w1
      { S7_Templates := "SrcType := DInt" } EQ_Contact(in1 := "Unit1.Em13.HmiInterface".jrUnloadingPnP.jobs.status.activeJobNumber, in2 := "U1EM13_JOB04")
      Coil( "ProdDataInterfaceHmi".cycleTimerDataSet[14].control[4].run )
   END_RUNG
   // the same network as SCL:
   "ProdDataInterfaceHmi".cycleTimerDataSet[14].control[1].run := #TRUE AND ("Unit1.Em13.HmiInterface".jrUnloadingPnP.jobs.status.activeJobNumber = "U1EM13_JOB01");
   "ProdDataInterfaceHmi".cycleTimerDataSet[14].control[2].run := #TRUE AND ("Unit1.Em13.HmiInterface".jrUnloadingPnP.jobs.status.activeJobNumber = "U1EM13_JOB02");
   "ProdDataInterfaceHmi".cycleTimerDataSet[14].control[3].run := #TRUE AND ("Unit1.Em13.HmiInterface".jrUnloadingPnP.jobs.status.activeJobNumber = "U1EM13_JOB03");
   "ProdDataInterfaceHmi".cycleTimerDataSet[14].control[4].run := #TRUE AND ("Unit1.Em13.HmiInterface".jrUnloadingPnP.jobs.status.activeJobNumber = "U1EM13_JOB04");
END_REGION
END_FUNCTION
